// TIA Portal V19 export
DATA_BLOCK "ProductionMng_PERS"   // DB16
// stored: MemoryReserve 100
   VAR RETAIN
      Pers { S7_SetPoint := 'True'} : "Prod_Pers";
   END_VAR
BEGIN
   Pers.Data.MODE.MES_ON := TRUE;
   Pers.Data.MODE.Cambio_Ordine_Automatico := TRUE;
   Pers.Data.SET_UP.Status := 10;
   Pers.Data.SET_UP.ProductionReady := TRUE;
   Pers.Data.SET_UP.Prepapration_Aut_Done_PPrf_Number := 201;
   Pers.Data.SET_UP.Prepapration_Man_Done_PPrf_Number := 201;
   Pers.Data.SET_UP.MSG101_inviato_MES_PPrf_Number := 201;
   Pers.Data.SET_UP.MSG101_inviato_LOG_PPrf_Number := 201;
   Pers.Data.SET_UP.MSG102_inviato_MES_PPrf_Number := 201;
   Pers.Data.SET_UP.MSG102_inviato_LOG_PPrf_Number := 201;
   Pers.Data.SET_UP.STS_Man_SetUp.Done := FALSE;
   Pers.Data.SET_UP.STS_Man_SetUp.Done_X := TRUE;
   Pers.Data.SET_UP.STS_Man_SetUp.Done_Y := TRUE;
   Pers.Data.SET_UP.STS_Man_SetUp.Done_Z := FALSE;
   Pers.Data.SET_UP.STS_Man_SetUp.Ack_Eseguito_X[1..50] := TRUE;
   Pers.Data.SET_UP.STS_Man_SetUp.Ack_Eseguito_Y[1..2] := TRUE;
   Pers.Data.SET_UP.STS_Man_SetUp.Ack_Eseguito_Y[3] := FALSE;
   Pers.Data.SET_UP.STS_Aut_SetUp.Assi_Profilatrice_InPosizione := TRUE;
   Pers.Data.SET_UP.STS_Aut_SetUp.Assi_Bordatrice_InPosizione := TRUE;
   Pers.Data.INTERRUZIONI.STOP_FineTurno := FALSE;
   Pers.Data.INTERRUZIONI.STOP_FineTurno_Done := FALSE;
   Pers.Data.INTERRUZIONI.STOP_ControlloQualita := FALSE;
   Pers.Data.INTERRUZIONI.STOP_ControlloQualita_Done := FALSE;
   Pers.Data.INTERRUZIONI.O_ACT.MES_IDP := 'Simula_C60x40x125_1000';
   Pers.Data.INTERRUZIONI.O_ACT.Halted_Cause.Code := 0;
   Pers.Data.INTERRUZIONI.O_ACT.Halted_Cause.Detail := '';
   Pers.Data.INTERRUZIONI.O_ACT.Last_Halted_Cause_Code := 0;
   Pers.Data.INTERRUZIONI.O_ACT.Mem_STOP := FALSE;
   Pers.Data.INTERRUZIONI.O_ENDING[1..5].MES_IDP := '';
   Pers.Data.INTERRUZIONI.O_ENDING[1..5].Halted_Cause.Code := 0;
   Pers.Data.INTERRUZIONI.O_ENDING[1..5].Halted_Cause.Detail := '';
   Pers.Data.INTERRUZIONI.O_ENDING[1].Last_Halted_Cause_Code := 3;
   Pers.Data.INTERRUZIONI.O_ENDING[2..5].Last_Halted_Cause_Code := 0;
   Pers.Data.INTERRUZIONI.O_ENDING[1..5].Stopped_MEM := 0;
   Pers.Data.Aspo_In_Linea_Prev_Values.C_ID := 2;
   Pers.Data.Aspo_In_Linea_Prev_Values.MES_IDP := 'Simula_C60x40x125_1000';
   Pers.Data.Aspo_In_Linea_Prev_Values.Decoiler_N := 1;
   Pers.Data.Aspo_In_Linea_Prev_Values.MES_CN := 'ffff';
   Pers.Data.Aspo_In_Linea_Prev_Values.MES_HN := 'dddd';
   Pers.Data.Aspo_In_Linea_Prev_Values.Stato_Rotolo := 3;
   Pers.Data.Aspo_In_Linea_Prev_Values.Provini_Richiesti := 1;
   Pers.Data.Aspo_In_Linea_Prev_Values.Provini_Eseguiti := 0;
   Pers.Data.Aspo_In_Linea_Prev_Values.Diametro_Rotolo := 500.0;
   Pers.Data.Aspo_In_Linea_Prev_Values.Spessore_Errore := 0;
   Pers.Data.Aspo_In_Linea_Prev_Values.Spessore_materiale_TEV := 0.0;
   Pers.Data.Aspo_In_Linea_Prev_Values.Spessore_Deroga_TKD := 0;
   Pers.Data.Aspo_In_Carico_Prev_Values.C_ID := 1;
   Pers.Data.Aspo_In_Carico_Prev_Values.MES_IDP := 'Simula_C60x40x125_1000';
   Pers.Data.Aspo_In_Carico_Prev_Values.Decoiler_N := 2;
   Pers.Data.Aspo_In_Carico_Prev_Values.MES_CN := 'aaaa';
   Pers.Data.Aspo_In_Carico_Prev_Values.MES_HN := 'bbbb';
   Pers.Data.Aspo_In_Carico_Prev_Values.Stato_Rotolo := 3;
   Pers.Data.Aspo_In_Carico_Prev_Values.Provini_Richiesti := 1;
   Pers.Data.Aspo_In_Carico_Prev_Values.Provini_Eseguiti := 1;
   Pers.Data.Aspo_In_Carico_Prev_Values.Diametro_Rotolo := 500.0;
   Pers.Data.Aspo_In_Carico_Prev_Values.Spessore_Errore := 0;
   Pers.Data.Aspo_In_Carico_Prev_Values.Spessore_materiale_TEV := 0.0;
   Pers.Data.Aspo_In_Carico_Prev_Values.Spessore_Deroga_TKD := 0;
   Pers.Data.Taglio_Finale_Prev_Values.C_ID := 1;
   Pers.Data.Taglio_Finale_Prev_Values.MES_IDP := 'Simula_C60x40x125_1000';
   Pers.Data.Taglio_Finale_Prev_Values.Decoiler_N := 0;
   Pers.Data.Taglio_Finale_Prev_Values.MES_CN := 'aaaa';
   Pers.Data.Taglio_Finale_Prev_Values.MES_HN := 'bbbb';
   Pers.Data.Taglio_Finale_Prev_Values.Stato_Rotolo := 0;
   Pers.Data.Taglio_Finale_Prev_Values.Provini_Richiesti := 0;
   Pers.Data.Taglio_Finale_Prev_Values.Provini_Eseguiti := 0;
   Pers.Data.Taglio_Finale_Prev_Values.Diametro_Rotolo := 0.0;
   Pers.Data.Taglio_Finale_Prev_Values.Spessore_Errore := 0;
   Pers.Data.Taglio_Finale_Prev_Values.Spessore_materiale_TEV := 0.0;
   Pers.Data.Taglio_Finale_Prev_Values.Spessore_Deroga_TKD := 0;
   Pers.Par.MES_Operating := 1;
   Pers.Par.AUT_PushOrder_InProduction := 1;
   Pers.Par.PartTolFactor_BAD_EXCEED_TOL := 3.0;
   Pers.Par.Material_To_Go_Additional := 10000.0;
   Pers.Par.Material_To_Go_Low_Speed := 4000.0;
END_DATA_BLOCK
